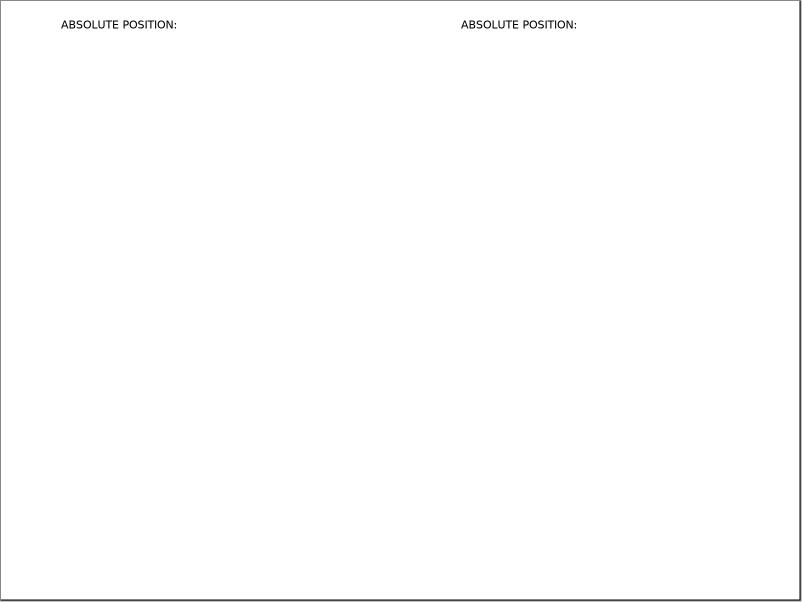
VISUALIZATION F21_Abort_Trigger  // 802x602
    Rectangle (0,0 800x600)
    Label (10,10 170x30), "ABSOLUTE POSITION:"
    Label (410,10 170x30), "ABSOLUTE POSITION:"
END_VISUALIZATION

(* stored: Version 1.1.0.1, ProductVersion 3.1.4022.7
   Visu F21_Abort_Trigger: Id {7c7458dc-91ff-44b7-9874-d7fe5fca15b7} *)
